// Two-queue serialized SDO reader for MCS2 channel parameters.
// Two independent state machines, both serializing onto the same slave but
// gated against each other so only one SDO request is outstanding at a time.
//
//   FAST queue: ChannelState only. Polled continuously at nReadTime. This is
//     the latency-sensitive path that interlocks depend on.
//
//   SLOW queue: the remaining 21 parameters (positioner type, calibration
//     options, sensor power mode, referencing options, reference type, safe
//     direction, motor load, channel type, max closed-loop frequency,
//     logical scale offset, logical scale inversion, channel temperature,
//     movement type, base unit, base resolution, distance code inverted,
//     positioner control options, actuator mode, motor load protection
//     threshold, diagnostic closed-loop frequency max and avg). Polled once
//     at boot,
//     then every nSlowReadTime (default 10 s). One read at a time. A failed
//     read logs / latches and the queue advances to the next entry.
//
// Both queues yield to each other: the fast queue will not start a new
// ChannelState read while the slow queue has one in flight, and vice versa.
// Because ChannelState reads are short (sub-100 ms) and the slow refresh
// cadence is ~10 s, ChannelState almost always wins the bus.

FUNCTION_BLOCK FB_ReadChanParameters
VAR_INPUT
    bEnable : BOOL;
END_VAR

VAR_IN_OUT
    stMotionStage       : ST_MotionStage;
    stMCS2ChanParameter : ST_MCS2ChanParameter;
    stDS402Drive        : ST_DS402Drive;
END_VAR

VAR_OUTPUT
    // TRUE once every entry in the slow queue has completed (succeeded or
    // failed) at least once. Diagnostic only -- not used to gate anything.
    bAllReadsComplete : BOOL;
    // Count of slow-queue entries that errored on their most recent attempt.
    // Cleared at the start of each slow sweep. Diagnostic only.
    nSlowReadFailures : UINT;
END_VAR

VAR

    // SDO reader instances

    // Fast queue
    fbChannelStateRead       : FB_EcCoESdoRead;
    // Event queue
    fbDriveErrCodeRead       : FB_EcCoESdoRead;
    // Slow queue
    fbMaxCloseLoopFreqRead   : FB_EcCoESdoRead;
    fbSoftLimMinRead         : FB_EcCoESdoRead;
    fbSoftLimMaxRead         : FB_EcCoESdoRead;
    fbPositionerTypeRead     : FB_EcCoESdoRead;
    fbCalibrationOptRead     : FB_EcCoESdoRead;
    fbSensorPowerModeRead    : FB_EcCoESdoRead;
    fbReferencingOptRead     : FB_EcCoESdoRead;
    fbReferenceTypeRead      : FB_EcCoESdoRead;
    fbSafeDirRead            : FB_EcCoESdoRead;
    fbMotorLoadRead          : FB_EcCoESdoRead;
    fbChannelTypeRead        : FB_EcCoESdoRead;
    fbLogicalScaleOffsetRead : FB_EcCoESdoRead;
    fbLogicalScaleInvRead    : FB_EcCoESdoRead;
    fbChannelTempRead        : FB_EcCoESdoRead;
    fbMovementTypeRead       : FB_EcCoESdoRead;
    fbBaseUnitRead           : FB_EcCoESdoRead;
    fbBaseResolutionRead     : FB_EcCoESdoRead;
    fbDistCodeInvRead        : FB_EcCoESdoRead;
    fbPositionerCtrlOptRead  : FB_EcCoESdoRead;
    fbActuatorModeRead       : FB_EcCoESdoRead;
    fbMotorLoadProtRead      : FB_EcCoESdoRead;
    // Diag closed-loop frequency is a subindexed object (0x202A:1 = max,
    // 0x202A:2 = avg); one reader per subindex.
    fbDiagClfMaxRead         : FB_EcCoESdoRead;
    fbDiagClfAvgRead         : FB_EcCoESdoRead;


    // Completion edge detectors

    ftChannelStateRead       : F_TRIG;
    ftDriveErrCodeRead       : F_TRIG;
    ftMaxCloseLoopFreqRead   : F_TRIG;
    ftSoftLimMinRead         : F_TRIG;
    ftSoftLimMaxRead         : F_TRIG;
    ftPositionerTypeRead     : F_TRIG;
    ftCalibrationOptRead     : F_TRIG;
    ftSensorPowerModeRead    : F_TRIG;
    ftReferencingOptRead     : F_TRIG;
    ftReferenceTypeRead      : F_TRIG;
    ftSafeDirRead            : F_TRIG;
    ftMotorLoadRead          : F_TRIG;
    ftChannelTypeRead        : F_TRIG;
    ftLogicalScaleOffsetRead : F_TRIG;
    ftLogicalScaleInvRead    : F_TRIG;
    ftChannelTempRead        : F_TRIG;
    ftMovementTypeRead       : F_TRIG;
    ftBaseUnitRead           : F_TRIG;
    ftBaseResolutionRead     : F_TRIG;
    ftDistCodeInvRead        : F_TRIG;
    ftPositionerCtrlOptRead  : F_TRIG;
    ftActuatorModeRead       : F_TRIG;
    ftMotorLoadProtRead      : F_TRIG;
    ftDiagClfMaxRead         : F_TRIG;
    ftDiagClfAvgRead         : F_TRIG;


    // Per-reader execute lines (driven by queue FSMs)

    bExecChannelState       : BOOL;
    bExecDriveErrCode       : BOOL;
    bExecMaxCloseLoopFreq   : BOOL;
    bExecSoftLimMin         : BOOL;
    bExecSoftLimMax         : BOOL;
    bExecPositionerType     : BOOL;
    bExecCalibrationOpt     : BOOL;
    bExecSensorPowerMode    : BOOL;
    bExecReferencingOpt     : BOOL;
    bExecReferenceType      : BOOL;
    bExecSafeDir            : BOOL;
    bExecMotorLoad          : BOOL;
    bExecChannelType        : BOOL;
    bExecLogicalScaleOffset : BOOL;
    bExecLogicalScaleInv    : BOOL;
    bExecChannelTemp        : BOOL;
    bExecMovementType       : BOOL;
    bExecBaseUnit           : BOOL;
    bExecBaseResolution     : BOOL;
    bExecDistCodeInv        : BOOL;
    bExecPositionerCtrlOpt  : BOOL;
    bExecActuatorMode       : BOOL;
    bExecMotorLoadProt      : BOOL;
    bExecDiagClfMax         : BOOL;
    bExecDiagClfAvg         : BOOL;


    // Fast queue (ChannelState)

    eFast : (
        FAST_IDLE          := 0,
        FAST_WAIT_CADENCE  := 1,
        FAST_READING       := 2
    ) := FAST_WAIT_CADENCE;
    tonFastCadence : TON;
    // Set on a fault or limit event: the drive error code reports the failed move,
    // not its cause, so the channel state bits must not be up to nReadTime stale.
    bFastReadNow : BOOL;
    // Per-read watchdog for ChannelState.
    tonFastReadTimeout : TON;
    tFastReadTimeout : TIME := T#2S;


    // Event queue (drive error code)

    // 0x603F holds the last channel error and is refreshed by the drive when the
    // Internal Limit flag is set, so it explains limit stops the NC cannot.
    eEvt : (
        EVT_IDLE    := 0,
        EVT_READING := 1
    ) := EVT_IDLE;
    rtErrEvent : R_TRIG;
    bEvtReadPending : BOOL;
    bEvtReadActive : BOOL;
    tonEvtReadTimeout : TON;
    tEvtReadTimeout : TIME := T#2S;


    // Slow queue (everything else)

    eSlow : (
        SLOW_IDLE       := 0,
        SLOW_WAIT_CADENCE := 1,
        SLOW_RUNNING    := 2
    ) := SLOW_IDLE;
    // Index into the slow-queue table. 1..NUM_SLOW; 0 = sweep complete.
    nSlowIdx : INT;
    // TRUE while a slow read is in flight (kick issued, edge not yet seen).
    bSlowReadActive : BOOL;
    tonSlowCadence : TON;
    // Per-read watchdog: if a slow read doesn't complete in tSlowReadTimeout
    // we count it as a failure, force-clear bExecute, and advance.
    tonSlowReadTimeout : TON;
    bFirstSlowSweepDone : BOOL;

    // Configurable cadences / timeouts for the slow queue.
    tSlowReadInterval : TIME := T#30S;
    tSlowReadTimeout  : TIME := T#2S;
END_VAR
VAR CONSTANT
    NUM_SLOW : INT := 23;
END_VAR

IF NOT __ISVALIDREF(stDS402Drive)
    OR NOT __ISVALIDREF(stMotionStage)
    OR NOT __ISVALIDREF(stMCS2ChanParameter) THEN
    RETURN;
END_IF

IF NOT bEnable THEN
    // Park everything off.
    bExecChannelState       := FALSE;
    bExecMaxCloseLoopFreq   := FALSE;
    bExecPositionerType     := FALSE;
    bExecCalibrationOpt     := FALSE;
    bExecSensorPowerMode    := FALSE;
    bExecReferencingOpt     := FALSE;
    bExecReferenceType      := FALSE;
    bExecSafeDir            := FALSE;
    bExecMotorLoad          := FALSE;
    bExecChannelType        := FALSE;
    bExecLogicalScaleOffset := FALSE;
    bExecLogicalScaleInv    := FALSE;
    bExecChannelTemp        := FALSE;
    bExecMovementType       := FALSE;
    bExecBaseUnit           := FALSE;
    bExecBaseResolution     := FALSE;
    bExecDistCodeInv        := FALSE;
    bExecPositionerCtrlOpt  := FALSE;
    bExecActuatorMode       := FALSE;
    bExecMotorLoadProt      := FALSE;
    bExecDiagClfMax         := FALSE;
    bExecDiagClfAvg         := FALSE;
    bExecDriveErrCode       := FALSE;
    bEvtReadPending         := FALSE;
    bEvtReadActive          := FALSE;
    bFastReadNow            := FALSE;
    eEvt                    := EVT_IDLE;
    tonEvtReadTimeout(IN := FALSE);
    tonFastCadence(IN := FALSE);
    tonSlowCadence(IN := FALSE);
    CallAllSdoReaders();
    RETURN;
END_IF

// Tick all the F_TRIGs from the previous cycle's bBusy snapshots.
ftChannelStateRead       (CLK := fbChannelStateRead.bBusy);
ftDriveErrCodeRead       (CLK := fbDriveErrCodeRead.bBusy);
ftMaxCloseLoopFreqRead   (CLK := fbMaxCloseLoopFreqRead.bBusy);
    ftSoftLimMinRead         (CLK := fbSoftLimMinRead.bBusy);
    ftSoftLimMaxRead         (CLK := fbSoftLimMaxRead.bBusy);
ftPositionerTypeRead     (CLK := fbPositionerTypeRead.bBusy);
ftCalibrationOptRead     (CLK := fbCalibrationOptRead.bBusy);
ftSensorPowerModeRead    (CLK := fbSensorPowerModeRead.bBusy);
ftReferencingOptRead     (CLK := fbReferencingOptRead.bBusy);
ftReferenceTypeRead      (CLK := fbReferenceTypeRead.bBusy);
ftSafeDirRead            (CLK := fbSafeDirRead.bBusy);
ftMotorLoadRead          (CLK := fbMotorLoadRead.bBusy);
ftChannelTypeRead        (CLK := fbChannelTypeRead.bBusy);
ftLogicalScaleOffsetRead (CLK := fbLogicalScaleOffsetRead.bBusy);
ftLogicalScaleInvRead    (CLK := fbLogicalScaleInvRead.bBusy);
ftChannelTempRead        (CLK := fbChannelTempRead.bBusy);
ftMovementTypeRead       (CLK := fbMovementTypeRead.bBusy);
ftBaseUnitRead           (CLK := fbBaseUnitRead.bBusy);
ftBaseResolutionRead     (CLK := fbBaseResolutionRead.bBusy);
ftDistCodeInvRead        (CLK := fbDistCodeInvRead.bBusy);
ftPositionerCtrlOptRead  (CLK := fbPositionerCtrlOptRead.bBusy);
ftActuatorModeRead       (CLK := fbActuatorModeRead.bBusy);
ftMotorLoadProtRead      (CLK := fbMotorLoadProtRead.bBusy);
ftDiagClfMaxRead         (CLK := fbDiagClfMaxRead.bBusy);
ftDiagClfAvgRead         (CLK := fbDiagClfAvgRead.bBusy);

// Run the two queues. Each yields to the other -- only one outstanding SDO
// at a time across the whole FB.
rtErrEvent(CLK := stMotionStage.bError OR stDS402Drive.stDriveStatus.InternalLimitActive);
IF rtErrEvent.Q THEN
    bEvtReadPending := TRUE;
    bFastReadNow    := TRUE;
END_IF

EventQueueStep();
FastQueueStep();
SlowQueueStep();

// Cyclically call every reader. bExecute lines are owned by the queues.
CallAllSdoReaders();

// Cyclic call of every SDO reader. Each FB's bExecute is owned by its queue.
METHOD PRIVATE CallAllSdoReaders
// Fast
fbChannelStateRead(
    sNetId     := stMotionStage.stAxisParameters.sAmsNetId,
    nSlaveAddr := stDS402Drive.nSlaveAddr,
    nIndex     := stMCS2ChanParameter.nChanStateIdx,
    nSubIndex  := 0,
    pDstBuf    := ADR(stMCS2ChanParameter.stChannelState.nChannelStateRaw),
    cbBufLen   := SIZEOF(stMCS2ChanParameter.stChannelState.nChannelStateRaw),
    bExecute   := bExecChannelState
);

// Event
fbDriveErrCodeRead(
    sNetId     := stMotionStage.stAxisParameters.sAmsNetId,
    nSlaveAddr := stDS402Drive.nSlaveAddr,
    nIndex     := stMCS2ChanParameter.nChanErrorCodeIdx,
    nSubIndex  := 0,
    pDstBuf    := ADR(stMCS2ChanParameter.nMCS2ErrorCode),
    cbBufLen   := SIZEOF(stMCS2ChanParameter.nMCS2ErrorCode),
    bExecute   := bExecDriveErrCode
);

// Slow
fbMaxCloseLoopFreqRead(
    sNetId     := stMotionStage.stAxisParameters.sAmsNetId,
    nSlaveAddr := stDS402Drive.nSlaveAddr,
    nIndex     := stMCS2ChanParameter.nChanMaxCloseLoopFreqIdx,
    nSubIndex  := 0,
    pDstBuf    := ADR(stMCS2ChanParameter.nMaxCloseLoopFreq),
    cbBufLen   := SIZEOF(stMCS2ChanParameter.nMaxCloseLoopFreq),
    bExecute   := bExecMaxCloseLoopFreq
);
fbSoftLimMinRead(
    sNetId     := stMotionStage.stAxisParameters.sAmsNetId,
    nSlaveAddr := stDS402Drive.nSlaveAddr,
    nIndex     := stMCS2ChanParameter.nChanSoftLimitIdx,
    nSubIndex  := 1,
    pDstBuf    := ADR(stMCS2ChanParameter.nSoftLimMin),
    cbBufLen   := SIZEOF(stMCS2ChanParameter.nSoftLimMin),
    bExecute   := bExecSoftLimMin
);
fbSoftLimMaxRead(
    sNetId     := stMotionStage.stAxisParameters.sAmsNetId,
    nSlaveAddr := stDS402Drive.nSlaveAddr,
    nIndex     := stMCS2ChanParameter.nChanSoftLimitIdx,
    nSubIndex  := 2,
    pDstBuf    := ADR(stMCS2ChanParameter.nSoftLimMax),
    cbBufLen   := SIZEOF(stMCS2ChanParameter.nSoftLimMax),
    bExecute   := bExecSoftLimMax
);
fbPositionerTypeRead(
    sNetId     := stMotionStage.stAxisParameters.sAmsNetId,
    nSlaveAddr := stDS402Drive.nSlaveAddr,
    nIndex     := stMCS2ChanParameter.nChanPositionerTypeIdx,
    nSubIndex  := 0,
    pDstBuf    := ADR(stMCS2ChanParameter.nPositionerType),
    cbBufLen   := SIZEOF(stMCS2ChanParameter.nPositionerType),
    bExecute   := bExecPositionerType
);
fbCalibrationOptRead(
    sNetId     := stMotionStage.stAxisParameters.sAmsNetId,
    nSlaveAddr := stDS402Drive.nSlaveAddr,
    nIndex     := stMCS2ChanParameter.nChanCalibrationOptIdx,
    nSubIndex  := 0,
    pDstBuf    := ADR(stMCS2ChanParameter.nCalibrationOpt),
    cbBufLen   := SIZEOF(stMCS2ChanParameter.nCalibrationOpt),
    bExecute   := bExecCalibrationOpt
);
fbSensorPowerModeRead(
    sNetId     := stMotionStage.stAxisParameters.sAmsNetId,
    nSlaveAddr := stDS402Drive.nSlaveAddr,
    nIndex     := stMCS2ChanParameter.nChanSensorPowerModeIdx,
    nSubIndex  := 0,
    pDstBuf    := ADR(stMCS2ChanParameter.nSensorPowerMode),
    cbBufLen   := SIZEOF(stMCS2ChanParameter.nSensorPowerMode),
    bExecute   := bExecSensorPowerMode
);
fbReferencingOptRead(
    sNetId     := stMotionStage.stAxisParameters.sAmsNetId,
    nSlaveAddr := stDS402Drive.nSlaveAddr,
    nIndex     := stMCS2ChanParameter.nChanReferencingOptIdx,
    nSubIndex  := 0,
    pDstBuf    := ADR(stMCS2ChanParameter.nReferencingOpt),
    cbBufLen   := SIZEOF(stMCS2ChanParameter.nReferencingOpt),
    bExecute   := bExecReferencingOpt
);
fbReferenceTypeRead(
    sNetId     := stMotionStage.stAxisParameters.sAmsNetId,
    nSlaveAddr := stDS402Drive.nSlaveAddr,
    nIndex     := stMCS2ChanParameter.nChanReferenceTypeIdx,
    nSubIndex  := 0,
    pDstBuf    := ADR(stMCS2ChanParameter.nReferenceType),
    cbBufLen   := SIZEOF(stMCS2ChanParameter.nReferenceType),
    bExecute   := bExecReferenceType
);
fbSafeDirRead(
    sNetId     := stMotionStage.stAxisParameters.sAmsNetId,
    nSlaveAddr := stDS402Drive.nSlaveAddr,
    nIndex     := stMCS2ChanParameter.nChanSafeDirIdx,
    nSubIndex  := 0,
    pDstBuf    := ADR(stMCS2ChanParameter.nSafeDir),
    cbBufLen   := SIZEOF(stMCS2ChanParameter.nSafeDir),
    bExecute   := bExecSafeDir
);
fbMotorLoadRead(
    sNetId     := stMotionStage.stAxisParameters.sAmsNetId,
    nSlaveAddr := stDS402Drive.nSlaveAddr,
    nIndex     := stMCS2ChanParameter.nChanMotorLoadIdx,
    nSubIndex  := 0,
    pDstBuf    := ADR(stMCS2ChanParameter.nMotorLoad),
    cbBufLen   := SIZEOF(stMCS2ChanParameter.nMotorLoad),
    bExecute   := bExecMotorLoad
);
fbChannelTypeRead(
    sNetId     := stMotionStage.stAxisParameters.sAmsNetId,
    nSlaveAddr := stDS402Drive.nSlaveAddr,
    nIndex     := stMCS2ChanParameter.nChannelTypeIdx,
    nSubIndex  := 0,
    pDstBuf    := ADR(stMCS2ChanParameter.nChannelType),
    cbBufLen   := SIZEOF(stMCS2ChanParameter.nChannelType),
    bExecute   := bExecChannelType
);
fbLogicalScaleOffsetRead(
    sNetId     := stMotionStage.stAxisParameters.sAmsNetId,
    nSlaveAddr := stDS402Drive.nSlaveAddr,
    nIndex     := stMCS2ChanParameter.nChanLogicalScaleOfsIdx,
    nSubIndex  := 0,
    pDstBuf    := ADR(stMCS2ChanParameter.nLogicalScaleOffset),
    cbBufLen   := SIZEOF(stMCS2ChanParameter.nLogicalScaleOffset),
    bExecute   := bExecLogicalScaleOffset
);
fbLogicalScaleInvRead(
    sNetId     := stMotionStage.stAxisParameters.sAmsNetId,
    nSlaveAddr := stDS402Drive.nSlaveAddr,
    nIndex     := stMCS2ChanParameter.nChanLogicalScaleInvIdx,
    nSubIndex  := 0,
    pDstBuf    := ADR(stMCS2ChanParameter.nLogicalScaleInv),
    cbBufLen   := SIZEOF(stMCS2ChanParameter.nLogicalScaleInv),
    bExecute   := bExecLogicalScaleInv
);
fbChannelTempRead(
    sNetId     := stMotionStage.stAxisParameters.sAmsNetId,
    nSlaveAddr := stDS402Drive.nSlaveAddr,
    nIndex     := stMCS2ChanParameter.nChanChannelTempIdx,
    nSubIndex  := 0,
    pDstBuf    := ADR(stMCS2ChanParameter.nChannelTemp),
    cbBufLen   := SIZEOF(stMCS2ChanParameter.nChannelTemp),
    bExecute   := bExecChannelTemp
);
fbMovementTypeRead(
    sNetId     := stMotionStage.stAxisParameters.sAmsNetId,
    nSlaveAddr := stDS402Drive.nSlaveAddr,
    nIndex     := stMCS2ChanParameter.nChanMovementTypeIdx,
    nSubIndex  := 0,
    pDstBuf    := ADR(stMCS2ChanParameter.nMovementType),
    cbBufLen   := SIZEOF(stMCS2ChanParameter.nMovementType),
    bExecute   := bExecMovementType
);
fbBaseUnitRead(
    sNetId     := stMotionStage.stAxisParameters.sAmsNetId,
    nSlaveAddr := stDS402Drive.nSlaveAddr,
    nIndex     := stMCS2ChanParameter.nChanBaseUnitIdx,
    nSubIndex  := 0,
    pDstBuf    := ADR(stMCS2ChanParameter.nBaseUnit),
    cbBufLen   := SIZEOF(stMCS2ChanParameter.nBaseUnit),
    bExecute   := bExecBaseUnit
);
fbBaseResolutionRead(
    sNetId     := stMotionStage.stAxisParameters.sAmsNetId,
    nSlaveAddr := stDS402Drive.nSlaveAddr,
    nIndex     := stMCS2ChanParameter.nChanBaseResolutionIdx,
    nSubIndex  := 0,
    pDstBuf    := ADR(stMCS2ChanParameter.nBaseResolution),
    cbBufLen   := SIZEOF(stMCS2ChanParameter.nBaseResolution),
    bExecute   := bExecBaseResolution
);
fbDistCodeInvRead(
    sNetId     := stMotionStage.stAxisParameters.sAmsNetId,
    nSlaveAddr := stDS402Drive.nSlaveAddr,
    nIndex     := stMCS2ChanParameter.nChanDistCodeInvIdx,
    nSubIndex  := 0,
    pDstBuf    := ADR(stMCS2ChanParameter.nDistCodeInv),
    cbBufLen   := SIZEOF(stMCS2ChanParameter.nDistCodeInv),
    bExecute   := bExecDistCodeInv
);
fbPositionerCtrlOptRead(
    sNetId     := stMotionStage.stAxisParameters.sAmsNetId,
    nSlaveAddr := stDS402Drive.nSlaveAddr,
    nIndex     := stMCS2ChanParameter.nChanPositionerCtrlOptIdx,
    nSubIndex  := 0,
    pDstBuf    := ADR(stMCS2ChanParameter.nPositionerCtrlOpt),
    cbBufLen   := SIZEOF(stMCS2ChanParameter.nPositionerCtrlOpt),
    bExecute   := bExecPositionerCtrlOpt
);
fbActuatorModeRead(
    sNetId     := stMotionStage.stAxisParameters.sAmsNetId,
    nSlaveAddr := stDS402Drive.nSlaveAddr,
    nIndex     := stMCS2ChanParameter.nChanActuatorModeIdx,
    nSubIndex  := 0,
    pDstBuf    := ADR(stMCS2ChanParameter.nActuatorMode),
    cbBufLen   := SIZEOF(stMCS2ChanParameter.nActuatorMode),
    bExecute   := bExecActuatorMode
);
fbMotorLoadProtRead(
    sNetId     := stMotionStage.stAxisParameters.sAmsNetId,
    nSlaveAddr := stDS402Drive.nSlaveAddr,
    nIndex     := stMCS2ChanParameter.nChanMotorLoadProtIdx,
    nSubIndex  := 0,
    pDstBuf    := ADR(stMCS2ChanParameter.nMotorLoadProt),
    cbBufLen   := SIZEOF(stMCS2ChanParameter.nMotorLoadProt),
    bExecute   := bExecMotorLoadProt
);
fbDiagClfMaxRead(
    sNetId     := stMotionStage.stAxisParameters.sAmsNetId,
    nSlaveAddr := stDS402Drive.nSlaveAddr,
    nIndex     := stMCS2ChanParameter.nChanDiagClfIdx,
    nSubIndex  := 1,
    pDstBuf    := ADR(stMCS2ChanParameter.nDiagClfMax),
    cbBufLen   := SIZEOF(stMCS2ChanParameter.nDiagClfMax),
    bExecute   := bExecDiagClfMax
);
fbDiagClfAvgRead(
    sNetId     := stMotionStage.stAxisParameters.sAmsNetId,
    nSlaveAddr := stDS402Drive.nSlaveAddr,
    nIndex     := stMCS2ChanParameter.nChanDiagClfIdx,
    nSubIndex  := 2,
    pDstBuf    := ADR(stMCS2ChanParameter.nDiagClfAvg),
    cbBufLen   := SIZEOF(stMCS2ChanParameter.nDiagClfAvg),
    bExecute   := bExecDiagClfAvg
);
END_METHOD

METHOD PRIVATE ClearAllSlowExecutes
bExecMaxCloseLoopFreq   := FALSE;
bExecPositionerType     := FALSE;
bExecCalibrationOpt     := FALSE;
bExecSensorPowerMode    := FALSE;
bExecReferencingOpt     := FALSE;
bExecReferenceType      := FALSE;
bExecSafeDir            := FALSE;
bExecMotorLoad          := FALSE;
bExecChannelType        := FALSE;
bExecLogicalScaleOffset := FALSE;
bExecLogicalScaleInv    := FALSE;
bExecChannelTemp        := FALSE;
bExecMovementType       := FALSE;
bExecBaseUnit           := FALSE;
bExecBaseResolution     := FALSE;
bExecDistCodeInv        := FALSE;
bExecPositionerCtrlOpt  := FALSE;
bExecActuatorMode       := FALSE;
bExecMotorLoadProt      := FALSE;
bExecDiagClfMax         := FALSE;
bExecDiagClfAvg         := FALSE;
bExecSoftLimMin         := FALSE;
bExecSoftLimMax         := FALSE;
END_METHOD

METHOD PRIVATE ClearSlowExecute
VAR_INPUT
    idx : INT;
END_VAR
CASE idx OF
    1:  bExecMaxCloseLoopFreq   := FALSE;
    2:  bExecPositionerType     := FALSE;
    3:  bExecCalibrationOpt     := FALSE;
    4:  bExecSensorPowerMode    := FALSE;
    5:  bExecReferencingOpt     := FALSE;
    6:  bExecReferenceType      := FALSE;
    7:  bExecSafeDir            := FALSE;
    8:  bExecMotorLoad          := FALSE;
    9:  bExecChannelType        := FALSE;
    10: bExecLogicalScaleOffset := FALSE;
    11: bExecLogicalScaleInv    := FALSE;
    12: bExecChannelTemp        := FALSE;
    13: bExecMovementType       := FALSE;
    14: bExecBaseUnit           := FALSE;
    15: bExecBaseResolution     := FALSE;
    16: bExecDistCodeInv        := FALSE;
    17: bExecPositionerCtrlOpt  := FALSE;
    18: bExecActuatorMode       := FALSE;
    19: bExecMotorLoadProt      := FALSE;
    20: bExecDiagClfMax         := FALSE;
    21: bExecDiagClfAvg         := FALSE;
    22: bExecSoftLimMin         := FALSE;
    23: bExecSoftLimMax         := FALSE;
END_CASE
END_METHOD

// Unpack the 32-bit raw channel state word into individual flag fields.
METHOD PRIVATE DecodeChannelState
VAR
    n : UDINT;
END_VAR
n := stMCS2ChanParameter.stChannelState.nChannelStateRaw;
stMCS2ChanParameter.stChannelState.bActivelyMoving        := (n AND 16#00000001) <> 0;
stMCS2ChanParameter.stChannelState.bClosedLoopActive      := (n AND 16#00000002) <> 0;
stMCS2ChanParameter.stChannelState.bCalibrating           := (n AND 16#00000004) <> 0;
stMCS2ChanParameter.stChannelState.bReferencing           := (n AND 16#00000008) <> 0;
stMCS2ChanParameter.stChannelState.bMoveDelayed           := (n AND 16#00000010) <> 0;
stMCS2ChanParameter.stChannelState.bSensorPresent         := (n AND 16#00000020) <> 0;
stMCS2ChanParameter.stChannelState.bIsCalibrated          := (n AND 16#00000040) <> 0;
stMCS2ChanParameter.stChannelState.bIsReferenced          := (n AND 16#00000080) <> 0;
stMCS2ChanParameter.stChannelState.bEndStopReached        := (n AND 16#00000100) <> 0;
stMCS2ChanParameter.stChannelState.bRangeLimitReached     := (n AND 16#00000200) <> 0;
stMCS2ChanParameter.stChannelState.bFollowingLimitReached := (n AND 16#00000400) <> 0;
stMCS2ChanParameter.stChannelState.bMovementFailed        := (n AND 16#00000800) <> 0;
stMCS2ChanParameter.stChannelState.bIsStreaming           := (n AND 16#00001000) <> 0;
stMCS2ChanParameter.stChannelState.bPositionerOverload    := (n AND 16#00002000) <> 0;
stMCS2ChanParameter.stChannelState.bOverTemperature       := (n AND 16#00004000) <> 0;
stMCS2ChanParameter.stChannelState.bReferenceMark         := (n AND 16#00008000) <> 0;
stMCS2ChanParameter.stChannelState.bIsPhased              := (n AND 16#00010000) <> 0;
stMCS2ChanParameter.stChannelState.bPositionerFault       := (n AND 16#00020000) <> 0;
stMCS2ChanParameter.stChannelState.bAmplifierEnabled      := (n AND 16#00040000) <> 0;
stMCS2ChanParameter.stChannelState.bInPosition            := (n AND 16#00080000) <> 0;
stMCS2ChanParameter.stChannelState.bBrakeEnabled          := (n AND 16#00100000) <> 0;
END_METHOD

// Event queue: one-shot read of the drive error code (0x603F) after a fault or
// internal-limit event. Highest priority, but still mutually exclusive with the
// fast and slow queues so only one SDO is outstanding on the mailbox.
METHOD PRIVATE EventQueueStep
CASE eEvt OF

    EVT_IDLE:
        bExecDriveErrCode := FALSE;
        bEvtReadActive    := FALSE;
        tonEvtReadTimeout(IN := FALSE);
        IF bEvtReadPending
           AND NOT bSlowReadActive
           AND (eFast <> FAST_READING) THEN
            bEvtReadPending   := FALSE;
            bExecDriveErrCode := TRUE;
            bEvtReadActive    := TRUE;
            eEvt              := EVT_READING;
        END_IF

    EVT_READING:
        tonEvtReadTimeout(IN := TRUE, PT := tEvtReadTimeout);
        IF ftDriveErrCodeRead.Q THEN
            // A failed read must not leave a stale code looking current.
            IF fbDriveErrCodeRead.bError THEN
                stMCS2ChanParameter.nMCS2ErrorCode := 0;
            END_IF
            bExecDriveErrCode := FALSE;
            bEvtReadActive    := FALSE;
            tonEvtReadTimeout(IN := FALSE);
            eEvt              := EVT_IDLE;
        ELSIF tonEvtReadTimeout.Q THEN
            stMCS2ChanParameter.nMCS2ErrorCode := 0;
            bExecDriveErrCode := FALSE;
            bEvtReadActive    := FALSE;
            tonEvtReadTimeout(IN := FALSE);
            eEvt              := EVT_IDLE;
        END_IF

END_CASE
END_METHOD

// Fast queue: poll ChannelState at nReadTime cadence. Yields the bus to the
// slow and event queues if one of those reads is currently in flight, but does
// not back off any further -- as soon as that read completes the fast read can fire.
METHOD PRIVATE FastQueueStep
CASE eFast OF

    FAST_IDLE:
        bExecChannelState := FALSE;
        eFast             := FAST_WAIT_CADENCE;

    FAST_WAIT_CADENCE:
        bExecChannelState := FALSE;
        tonFastReadTimeout(IN := FALSE);
        // Cadence timer runs while we're waiting for our next turn.
        tonFastCadence(
            IN := stMotionStage.bAxisParamsInit,
            PT := stMCS2ChanParameter.nReadTime
        );
        // Only fire when the cadence has elapsed AND the slow queue isn't
        // currently using the mailbox.
        IF (tonFastCadence.Q OR bFastReadNow) AND NOT bSlowReadActive AND NOT bEvtReadActive THEN
            tonFastCadence(IN := FALSE);
            bFastReadNow      := FALSE;
            bExecChannelState := TRUE;
            eFast             := FAST_READING;
        END_IF

    FAST_READING:
        // Hold execute TRUE through the read. F_TRIG on bBusy falling = done.
        tonFastReadTimeout(IN := TRUE, PT := tFastReadTimeout);
        IF ftChannelStateRead.Q THEN
            IF NOT fbChannelStateRead.bError THEN
                DecodeChannelState();
            ELSE
                // Don't stop polling on a single failure. Log once per
                // failure if motion subsystem isn't already noisy.
                IF NOT stMotionStage.bBusy THEN
                    stMotionStage.sErrorMessage := 'Failed to read ChannelState';
                END_IF
            END_IF
            bExecChannelState := FALSE;
            tonFastReadTimeout(IN := FALSE);
            eFast             := FAST_WAIT_CADENCE;
        ELSIF tonFastReadTimeout.Q THEN
            // Hung read -- give up and retry next cadence.
            IF NOT stMotionStage.bBusy THEN
                stMotionStage.sErrorMessage := 'ChannelState read timeout';
            END_IF
            bExecChannelState := FALSE;
            tonFastReadTimeout(IN := FALSE);
            eFast             := FAST_WAIT_CADENCE;
        END_IF

END_CASE
END_METHOD

// Slow queue: sweep through 21 entries once at boot, then refresh every
// tSlowReadInterval. One entry at a time. A failed read latches a counter
// and advances -- it does not stall the sweep or affect the fast queue.
METHOD PRIVATE SlowQueueStep
CASE eSlow OF

    SLOW_IDLE:
        ClearAllSlowExecutes();
        bSlowReadActive := FALSE;
        // Begin first sweep as soon as axis params are initialized.
        IF stMotionStage.bAxisParamsInit THEN
            nSlowIdx          := 1;
            nSlowReadFailures := 0;
            eSlow             := SLOW_RUNNING;
        END_IF

    SLOW_WAIT_CADENCE:
        ClearAllSlowExecutes();
        bSlowReadActive := FALSE;
        tonSlowCadence(
            IN := stMotionStage.bAxisParamsInit,
            PT := tSlowReadInterval
        );
        IF tonSlowCadence.Q THEN
            tonSlowCadence(IN := FALSE);
            nSlowIdx          := 1;
            nSlowReadFailures := 0;
            eSlow             := SLOW_RUNNING;
        END_IF

    SLOW_RUNNING:
        // Yield: never start a new slow read while the fast queue is
        // mid-read. Existing in-flight slow reads continue.
        IF NOT bSlowReadActive AND ((eFast = FAST_READING) OR bEvtReadActive) THEN
            // Just hold; don't kick the next read yet.
            RETURN;
        END_IF

        IF NOT bSlowReadActive THEN
            // Start the read at the current index.
            StartSlowRead(nSlowIdx);
            bSlowReadActive := TRUE;
            tonSlowReadTimeout(IN := FALSE);   // reset
        ELSE
            // Arm watchdog while we wait.
            tonSlowReadTimeout(IN := TRUE, PT := tSlowReadTimeout);
            IF SlowReadEdge(nSlowIdx) THEN
                // Normal completion path.
                IF SlowReadError(nSlowIdx) THEN
                    nSlowReadFailures := nSlowReadFailures + 1;
                END_IF
                ClearSlowExecute(nSlowIdx);
                bSlowReadActive := FALSE;
                tonSlowReadTimeout(IN := FALSE);
                nSlowIdx := nSlowIdx + 1;
            ELSIF tonSlowReadTimeout.Q THEN
                // Hung read -- force-clear and advance. The reader FB will
                // see bExecute drop; whether it ever asserts an edge later
                // is its problem, not ours.
                nSlowReadFailures := nSlowReadFailures + 1;
                ClearSlowExecute(nSlowIdx);
                bSlowReadActive := FALSE;
                tonSlowReadTimeout(IN := FALSE);
                nSlowIdx := nSlowIdx + 1;
            END_IF

            IF nSlowIdx > NUM_SLOW THEN
                // Sweep done.
                bFirstSlowSweepDone := TRUE;
                bAllReadsComplete   := TRUE;
                nSlowIdx            := 0;
                eSlow               := SLOW_WAIT_CADENCE;
            END_IF
        END_IF

END_CASE
END_METHOD

// Return TRUE on the cycle the read at <idx> completes (busy->idle).
METHOD PRIVATE SlowReadEdge : BOOL
VAR_INPUT
    idx : INT;
END_VAR
CASE idx OF
    1:  SlowReadEdge := ftMaxCloseLoopFreqRead.Q;
    2:  SlowReadEdge := ftPositionerTypeRead.Q;
    3:  SlowReadEdge := ftCalibrationOptRead.Q;
    4:  SlowReadEdge := ftSensorPowerModeRead.Q;
    5:  SlowReadEdge := ftReferencingOptRead.Q;
    6:  SlowReadEdge := ftReferenceTypeRead.Q;
    7:  SlowReadEdge := ftSafeDirRead.Q;
    8:  SlowReadEdge := ftMotorLoadRead.Q;
    9:  SlowReadEdge := ftChannelTypeRead.Q;
    10: SlowReadEdge := ftLogicalScaleOffsetRead.Q;
    11: SlowReadEdge := ftLogicalScaleInvRead.Q;
    12: SlowReadEdge := ftChannelTempRead.Q;
    13: SlowReadEdge := ftMovementTypeRead.Q;
    14: SlowReadEdge := ftBaseUnitRead.Q;
    15: SlowReadEdge := ftBaseResolutionRead.Q;
    16: SlowReadEdge := ftDistCodeInvRead.Q;
    17: SlowReadEdge := ftPositionerCtrlOptRead.Q;
    18: SlowReadEdge := ftActuatorModeRead.Q;
    19: SlowReadEdge := ftMotorLoadProtRead.Q;
    20: SlowReadEdge := ftDiagClfMaxRead.Q;
    21: SlowReadEdge := ftDiagClfAvgRead.Q;
    22: SlowReadEdge := ftSoftLimMinRead.Q;
    23: SlowReadEdge := ftSoftLimMaxRead.Q;
    ELSE
        SlowReadEdge := FALSE;
END_CASE
END_METHOD

// Return the .bError flag for the read at <idx> after completion.
METHOD PRIVATE SlowReadError : BOOL
VAR_INPUT
    idx : INT;
END_VAR
CASE idx OF
    1:  SlowReadError := fbMaxCloseLoopFreqRead.bError;
    2:  SlowReadError := fbPositionerTypeRead.bError;
    3:  SlowReadError := fbCalibrationOptRead.bError;
    4:  SlowReadError := fbSensorPowerModeRead.bError;
    5:  SlowReadError := fbReferencingOptRead.bError;
    6:  SlowReadError := fbReferenceTypeRead.bError;
    7:  SlowReadError := fbSafeDirRead.bError;
    8:  SlowReadError := fbMotorLoadRead.bError;
    9:  SlowReadError := fbChannelTypeRead.bError;
    10: SlowReadError := fbLogicalScaleOffsetRead.bError;
    11: SlowReadError := fbLogicalScaleInvRead.bError;
    12: SlowReadError := fbChannelTempRead.bError;
    13: SlowReadError := fbMovementTypeRead.bError;
    14: SlowReadError := fbBaseUnitRead.bError;
    15: SlowReadError := fbBaseResolutionRead.bError;
    16: SlowReadError := fbDistCodeInvRead.bError;
    17: SlowReadError := fbPositionerCtrlOptRead.bError;
    18: SlowReadError := fbActuatorModeRead.bError;
    19: SlowReadError := fbMotorLoadProtRead.bError;
    20: SlowReadError := fbDiagClfMaxRead.bError;
    21: SlowReadError := fbDiagClfAvgRead.bError;
    22: SlowReadError := fbSoftLimMinRead.bError;
    23: SlowReadError := fbSoftLimMaxRead.bError;
    ELSE
        SlowReadError := FALSE;
END_CASE
END_METHOD

// Issue bExecute=TRUE for the slow-queue entry at the given index.
METHOD PRIVATE StartSlowRead
VAR_INPUT
    idx : INT;
END_VAR
CASE idx OF
    1:  bExecMaxCloseLoopFreq   := TRUE;
    2:  bExecPositionerType     := TRUE;
    3:  bExecCalibrationOpt     := TRUE;
    4:  bExecSensorPowerMode    := TRUE;
    5:  bExecReferencingOpt     := TRUE;
    6:  bExecReferenceType      := TRUE;
    7:  bExecSafeDir            := TRUE;
    8:  bExecMotorLoad          := TRUE;
    9:  bExecChannelType        := TRUE;
    10: bExecLogicalScaleOffset := TRUE;
    11: bExecLogicalScaleInv    := TRUE;
    12: bExecChannelTemp        := TRUE;
    13: bExecMovementType       := TRUE;
    14: bExecBaseUnit           := TRUE;
    15: bExecBaseResolution     := TRUE;
    16: bExecDistCodeInv        := TRUE;
    17: bExecPositionerCtrlOpt  := TRUE;
    18: bExecActuatorMode       := TRUE;
    19: bExecMotorLoadProt      := TRUE;
    20: bExecDiagClfMax         := TRUE;
    21: bExecDiagClfAvg         := TRUE;
    22: bExecSoftLimMin         := TRUE;
    23: bExecSoftLimMax         := TRUE;
END_CASE
END_METHOD

END_FUNCTION_BLOCK

(* stored: Version 1.1.0.1
   POU FB_ReadChanParameters: Id {08ee74cb-7e7d-468d-8ff5-637be4dc44de}, SpecialFunc None
   Method CallAllSdoReaders: Id {0a000001-0000-0000-0000-000000000009}
   Method ClearAllSlowExecutes: Id {0a000001-0000-0000-0000-000000000005}
   Method ClearSlowExecute: Id {0a000001-0000-0000-0000-000000000004}
   Method DecodeChannelState: Id {0a000001-0000-0000-0000-000000000008}
   Method EventQueueStep: Id {0a000001-0000-0000-0000-00000000000a}
   Method FastQueueStep: Id {0a000001-0000-0000-0000-000000000001}
   Method SlowQueueStep: Id {0a000001-0000-0000-0000-000000000002}
   Method SlowReadEdge: Id {0a000001-0000-0000-0000-000000000006}
   Method SlowReadError: Id {0a000001-0000-0000-0000-000000000007}
   Method StartSlowRead: Id {0a000001-0000-0000-0000-000000000003} *)
